TYPE ST_CoolingControlHmi :
STRUCT
	// HMI -> PLC
	sName					: STRING;
	paramRoomTempSet		: REAL;
	param_P					: REAL;
	param_I					: REAL;
	Param_D					: REAL;
	
	nMotorManualSpeed		: INT;
END_STRUCT
END_TYPE

(* stored: Version 1.1.0.1
   DUT ST_CoolingControlHmi: Id {04931081-96f2-4cd7-8d65-b2759124a6c0} *)
